INTERFACE IEventHandlerBase EXTENDS __SYSTEM.IQueryInterface

END_INTERFACE

(* stored: Version 1.1.0.1, ProductVersion 3.1.4024.3
   Itf IEventHandlerBase: Id {2c3ca761-e7a8-0b83-1e2e-ea427463059e} *)
